  933 | Hüllkurvensteuerung: Mindestgrenze für Hochdruck des Verdichters 3 „Wie oben, für den Verdichter Nr.3“. M CO | Hüllkurvensteuerung: Mindestgrenze für Hochdruck des Verdichters 3 „Wie oben, für den Verdichter Nr.3“. M CO | Envelope control: Mindestgrenze für Hochdruck compressors 3 „Wie oben, für compressor Nr.3“. M CO | Envelope control: Mindestgrenze für Hochdruck compresseurs 3 „Wie oben, für compresseur Nr.3“. M CO | Envelope control: Mindestgrenze für Hochdruck compressores 3 „Wie oben, für compressore Nr.3“. M CO
  934 | Hüllkurvensteuerung: Mindestgrenze für Hochdruck des Verdichters 4 „Wie oben, für den Verdichter Nr.4“. M CO | Hüllkurvensteuerung: Mindestgrenze für Hochdruck des Verdichters 4 „Wie oben, für den Verdichter Nr.4“. M CO | Envelope control: Mindestgrenze für Hochdruck compressors 4 „Wie oben, für compressor Nr.4“. M CO | Envelope control: Mindestgrenze für Hochdruck compresseurs 4 „Wie oben, für compresseur Nr.4“. M CO | Envelope control: Mindestgrenze für Hochdruck compressores 4 „Wie oben, für compressore Nr.4“. M CO
  935 | Hüllkurvensteuerung: Mindestgrenze für Hochdruck des Verdichters 5 „Wie oben, für den Verdichter Nr. 5“. M CO | Hüllkurvensteuerung: Mindestgrenze für Hochdruck des Verdichters 5 „Wie oben, für den Verdichter Nr. 5“. M CO | Envelope control: Mindestgrenze für Hochdruck compressors 5 „Wie oben, für compressor Nr. 5“. M CO | Envelope control: Mindestgrenze für Hochdruck compresseurs 5 „Wie oben, für compresseur Nr. 5“. M CO | Envelope control: Mindestgrenze für Hochdruck compressores 5 „Wie oben, für compressore Nr. 5“. M CO
  936 | Hüllkurvensteuerung: Mindestgrenze für Hochdruck des Verdichters 6 „Wie oben, für den Verdichter Nr. 6“. M CO | Hüllkurvensteuerung: Mindestgrenze für Hochdruck des Verdichters 6 „Wie oben, für den Verdichter Nr. 6“. M CO | Envelope control: Mindestgrenze für Hochdruck compressors 6 „Wie oben, für compressor Nr. 6“. M CO | Envelope control: Mindestgrenze für Hochdruck compresseurs 6 „Wie oben, für compresseur Nr. 6“. M CO | Envelope control: Mindestgrenze für Hochdruck compressores 6 „Wie oben, für compressore Nr. 6“. M CO
  937 | Hüllkurvensteuerung: Mindestgrenze für Hochdruck des Verdichters 7 „Wie oben, für den Verdichter Nr. 7“. M CO | Hüllkurvensteuerung: Mindestgrenze für Hochdruck des Verdichters 7 „Wie oben, für den Verdichter Nr. 7“. M CO | Envelope control: Mindestgrenze für Hochdruck compressors 7 „Wie oben, für compressor Nr. 7“. M CO | Envelope control: Mindestgrenze für Hochdruck compresseurs 7 „Wie oben, für compresseur Nr. 7“. M CO | Envelope control: Mindestgrenze für Hochdruck compressores 7 „Wie oben, für compressore Nr. 7“. M CO
  938 | Hüllkurvensteuerung: Mindestgrenze für Hochdruck des Verdichters 8 „Wie oben, für den Verdichter Nr. 8“. M CO | Hüllkurvensteuerung: Mindestgrenze für Hochdruck des Verdichters 8 „Wie oben, für den Verdichter Nr. 8“. M CO | Envelope control: Mindestgrenze für Hochdruck compressors 8 „Wie oben, für compressor Nr. 8“. M CO | Envelope control: Mindestgrenze für Hochdruck compresseurs 8 „Wie oben, für compresseur Nr. 8“. M CO | Envelope control: Mindestgrenze für Hochdruck compressores 8 „Wie oben, für compressore Nr. 8“. M CO
  941 | Min. Verdichtungsverhältnis beim Anlaufen des Verdichters 1 | Min. Verdichtungsverhältnis beim Anlaufen des Verdichters 1 | Min. Verdichtungsverhältnis beim Anlaufen compressors 1 | Min. Verdichtungsverhältnis beim Anlaufen compresseurs 1 | Min. Verdichtungsverhältnis beim Anlaufen compressores 1
  942 | Min. Verdichtungsverhältnis beim Anlaufen des Verdichters 2 „Wie oben, für den Verdichter Nr.2“. M CO | Min. Verdichtungsverhältnis beim Anlaufen des Verdichters 2 „Wie oben, für den Verdichter Nr.2“. M CO | Min. Verdichtungsverhältnis beim Anlaufen compressors 2 „Wie oben, für compressor Nr.2“. M CO | Min. Verdichtungsverhältnis beim Anlaufen compresseurs 2 „Wie oben, für compresseur Nr.2“. M CO | Min. Verdichtungsverhältnis beim Anlaufen compressores 2 „Wie oben, für compressore Nr.2“. M CO
  943 | Min. Verdichtungsverhältnis beim Anlaufen des Verdichters 3 „Wie oben, für den Verdichter Nr.3“. M CO | Min. Verdichtungsverhältnis beim Anlaufen des Verdichters 3 „Wie oben, für den Verdichter Nr.3“. M CO | Min. Verdichtungsverhältnis beim Anlaufen compressors 3 „Wie oben, für compressor Nr.3“. M CO | Min. Verdichtungsverhältnis beim Anlaufen compresseurs 3 „Wie oben, für compresseur Nr.3“. M CO | Min. Verdichtungsverhältnis beim Anlaufen compressores 3 „Wie oben, für compressore Nr.3“. M CO
  944 | Min. Verdichtungsverhältnis beim Anlaufen des Verdichters 4 „Wie oben, für den Verdichter Nr.4“. M CO | Min. Verdichtungsverhältnis beim Anlaufen des Verdichters 4 „Wie oben, für den Verdichter Nr.4“. M CO | Min. Verdichtungsverhältnis beim Anlaufen compressors 4 „Wie oben, für compressor Nr.4“. M CO | Min. Verdichtungsverhältnis beim Anlaufen compresseurs 4 „Wie oben, für compresseur Nr.4“. M CO | Min. Verdichtungsverhältnis beim Anlaufen compressores 4 „Wie oben, für compressore Nr.4“. M CO
  945 | Min. Verdichtungsverhältnis beim Anlaufen des Verdichters 5 „Wie oben, für den Verdichter Nr. 5“. M CO | Min. Verdichtungsverhältnis beim Anlaufen des Verdichters 5 „Wie oben, für den Verdichter Nr. 5“. M CO | Min. Verdichtungsverhältnis beim Anlaufen compressors 5 „Wie oben, für compressor Nr. 5“. M CO | Min. Verdichtungsverhältnis beim Anlaufen compresseurs 5 „Wie oben, für compresseur Nr. 5“. M CO | Min. Verdichtungsverhältnis beim Anlaufen compressores 5 „Wie oben, für compressore Nr. 5“. M CO
  946 | Min. Verdichtungsverhältnis beim Anlaufen des Verdichters 6 „Wie oben, für den Verdichter Nr. 6“. M CO | Min. Verdichtungsverhältnis beim Anlaufen des Verdichters 6 „Wie oben, für den Verdichter Nr. 6“. M CO | Min. Verdichtungsverhältnis beim Anlaufen compressors 6 „Wie oben, für compressor Nr. 6“. M CO | Min. Verdichtungsverhältnis beim Anlaufen compresseurs 6 „Wie oben, für compresseur Nr. 6“. M CO | Min. Verdichtungsverhältnis beim Anlaufen compressores 6 „Wie oben, für compressore Nr. 6“. M CO
  947 | Min. Verdichtungsverhältnis beim Anlaufen des Verdichters 7 „Wie oben, für den Verdichter Nr. 7“. M CO | Min. Verdichtungsverhältnis beim Anlaufen des Verdichters 7 „Wie oben, für den Verdichter Nr. 7“. M CO | Min. Verdichtungsverhältnis beim Anlaufen compressors 7 „Wie oben, für compressor Nr. 7“. M CO | Min. Verdichtungsverhältnis beim Anlaufen compresseurs 7 „Wie oben, für compresseur Nr. 7“. M CO | Min. Verdichtungsverhältnis beim Anlaufen compressores 7 „Wie oben, für compressore Nr. 7“. M CO
  948 | Min. Verdichtungsverhältnis beim Anlaufen des Verdichters 8 „Wie oben, für den Verdichter Nr. 8“. M CO | Min. Verdichtungsverhältnis beim Anlaufen des Verdichters 8 „Wie oben, für den Verdichter Nr. 8“. M CO | Min. Verdichtungsverhältnis beim Anlaufen compressors 8 „Wie oben, für compressor Nr. 8“. M CO | Min. Verdichtungsverhältnis beim Anlaufen compresseurs 8 „Wie oben, für compresseur Nr. 8“. M CO | Min. Verdichtungsverhältnis beim Anlaufen compressores 8 „Wie oben, für compressore Nr. 8“. M CO
  951 | Trennung HGBP -Ventil des Verdichters 1 | Trennung HGBP -Ventil des Verdichters 1 | Disconnection HGBP -Ventil compressors 1 | Disconnection HGBP -Ventil compresseurs 1 | Disconnection HGBP -Ventil compressores 1
  952 | Trennung HGBP -Ventil des Verdichters 2 „Wie oben, für den Verdichter Nr.2“. S CO | Trennung HGBP -Ventil des Verdichters 2 „Wie oben, für den Verdichter Nr.2“. S CO | Disconnection HGBP -Ventil compressors 2 „Wie oben, für compressor Nr.2“. S CO | Disconnection HGBP -Ventil compresseurs 2 „Wie oben, für compresseur Nr.2“. S CO | Disconnection HGBP -Ventil compressores 2 „Wie oben, für compressore Nr.2“. S CO
  953 | Trennung HGBP -Ventil des Verdichters 3 „Wie oben, für den Verdichter Nr.3“. S CO | Trennung HGBP -Ventil des Verdichters 3 „Wie oben, für den Verdichter Nr.3“. S CO | Disconnection HGBP -Ventil compressors 3 „Wie oben, für compressor Nr.3“. S CO | Disconnection HGBP -Ventil compresseurs 3 „Wie oben, für compresseur Nr.3“. S CO | Disconnection HGBP -Ventil compressores 3 „Wie oben, für compressore Nr.3“. S CO
  954 | Trennung HGBP -Ventil des Verdichters 4 „Wie oben, für den Verdichter Nr.4“. S CO | Trennung HGBP -Ventil des Verdichters 4 „Wie oben, für den Verdichter Nr.4“. S CO | Disconnection HGBP -Ventil compressors 4 „Wie oben, für compressor Nr.4“. S CO | Disconnection HGBP -Ventil compresseurs 4 „Wie oben, für compresseur Nr.4“. S CO | Disconnection HGBP -Ventil compressores 4 „Wie oben, für compressore Nr.4“. S CO
  960 | Trennung thermal meter | Trennung thermal meter | Disconnection thermal meter | Disconnection thermal meter | Disconnection thermal meter
  961 | Offline Driver erste Stufe Nr.5 | Offline Driver erste Stufe Nr.5 | Offline Driver erste Stufe Nr.5 | Offline Driver erste Stufe Nr.5 | Offline Driver erste Stufe Nr.5
  962 | Offline Driver erste Stufe Nr.6 „Wie oben, für den Verdichter 6“. A CI | Offline Driver erste Stufe Nr.6 „Wie oben, für den Verdichter 6“. A CI | Offline Driver erste Stufe Nr.6 „Wie oben, für compressor 6“. A CI | Offline Driver erste Stufe Nr.6 „Wie oben, für compresseur 6“. A CI | Offline Driver erste Stufe Nr.6 „Wie oben, für compressore 6“. A CI
  963 | Offline Driver erste Stufe Nr.7 „Wie oben, für den Verdichter 7“. A CI | Offline Driver erste Stufe Nr.7 „Wie oben, für den Verdichter 7“. A CI | Offline Driver erste Stufe Nr.7 „Wie oben, für compressor 7“. A CI | Offline Driver erste Stufe Nr.7 „Wie oben, für compresseur 7“. A CI | Offline Driver erste Stufe Nr.7 „Wie oben, für compressore 7“. A CI
  964 | Offline Driver erste Stufe Nr.8 „Wie oben, für den Verdichter 8“. A CI | Offline Driver erste Stufe Nr.8 „Wie oben, für den Verdichter 8“. A CI | Offline Driver erste Stufe Nr.8 „Wie oben, für compressor 8“. A CI | Offline Driver erste Stufe Nr.8 „Wie oben, für compresseur 8“. A CI | Offline Driver erste Stufe Nr.8 „Wie oben, für compressore 8“. A CI
  965 | Trennung ATS | Trennung ATS | Disconnection ATS | Disconnection ATS | Disconnection ATS
  966 | Trennung Touch HT -Zone Meldet die Trennung des Touch -Thermostaten der Zone HT. S GR | Trennung Touch HT -Zone Meldet die Trennung des Touch -Thermostaten der Zone HT. S GR | Disconnection Touch HT -Zone Meldet Trennung Touch -Thermostaten Zone HT. S GR | Disconnection Touch HT -Zone Meldet Trennung Touch -Thermostaten Zone HT. S GR | Disconnection Touch HT -Zone Meldet Trennung Touch -Thermostaten Zone HT. S GR
  967 | Trennung Touch LT -Zone Meldet die Trennung des Touch -Thermostaten der Zone LT. S GR | Trennung Touch LT -Zone Meldet die Trennung des Touch -Thermostaten der Zone LT. S GR | Disconnection Touch LT -Zone Meldet Trennung Touch -Thermostaten Zone LT. S GR | Disconnection Touch LT -Zone Meldet Trennung Touch -Thermostaten Zone LT. S GR | Disconnection Touch LT -Zone Meldet Trennung Touch -Thermostaten Zone LT. S GR
  968 | Verhinderung von Stillstand des Verdichters Meldet die Zwangsabschaltung des Inverter - Verdichters und seines Kreislaufs, um einen Stillstand aufgrund eines zu hohen Stromverbrauchs zu verhindern. M CI | Verhinderung von Stillstand des Verdichters Meldet die Zwangsabschaltung des Inverter - Verdichters und seines Kreislaufs, um einen Stillstand aufgrund eines zu hohen Stromverbrauchs zu verhindern. M CI | Verhinderung von Stillstand compressors Meldet Zwangsabschaltung inverter - compressors und seines circuits, um einen Stillstand aufgrund eines zu hohen Stromverbrauchs zu verhindern. M CI | Verhinderung von Stillstand compresseurs Meldet Zwangsabschaltung variateur - compresseurs und seines circuits, um einen Stillstand aufgrund eines zu hohen Stromverbrauchs zu verhindern. M CI | Verhinderung von Stillstand compressores Meldet Zwangsabschaltung inverter - compressores und seines circuitos, um einen Stillstand aufgrund eines zu hohen Stromverbrauchs zu verhindern. M CI
  969 | Hohe Außenlufttemperatur Meldet, dass das Gerät bei einer zu hohen Außentemperatur betrieben wird. Die Kontrolle erfolgt auch bei ausgeschalteten Verdichtern. S-M U STG0200 | Hohe Außenlufttemperatur Meldet, dass das Gerät bei einer zu hohen Außentemperatur betrieben wird. Die Kontrolle erfolgt auch bei ausgeschalteten Verdichtern. S-M U STG0200 | Hohe outdoor air temperature Meldet, dass Gerät bei einer zu hohen Außentemperatur betrieben wird. Kontrolle erfolgt auch bei ausgeschalteten compressorn. S-M U STG0200 | Hohe température extérieure Meldet, dass Gerät bei einer zu hohen Außentemperatur betrieben wird. Kontrolle erfolgt auch bei ausgeschalteten compresseurn. S-M U STG0200 | Hohe temperatura aria esterna Meldet, dass Gerät bei einer zu hohen Außentemperatur betrieben wird. Kontrolle erfolgt auch bei ausgeschalteten compressoren. S-M U STG0200
  970 | Geringer Wassergehalt bei der Wärmerückgewinnung. Meldet einen Wassermangel im Wasserkreislauf für die Wärmerückgewinnung. Dieser Mangel führt zu plötzlichen Wechseln der Betriebsart der Kreisläufe, wodurch die Ventile des Kältemittelkreislaufs beschädigt werden können. S-M U | Geringer Wassergehalt bei der Wärmerückgewinnung. Meldet einen Wassermangel im Wasserkreislauf für die Wärmerückgewinnung. Dieser Mangel führt zu plötzlichen Wechseln der Betriebsart der Kreisläufe, wodurch die Ventile des Kältemittelkreislaufs beschädigt werden können. S-M U | Geringer Wassergehalt bei heat recovery. Meldet einen Wassermangel im Wassercircuit für heat recovery. Dieser Mangel führt zu plötzlichen Wechseln Betriebsart Kreisläufe, wodurch Ventile Kältemittelcircuits beschädigt werden können. S-M U | Geringer Wassergehalt bei récupération de chaleur. Meldet einen Wassermangel im Wassercircuit für récupération de chaleur. Dieser Mangel führt zu plötzlichen Wechseln Betriebsart Kreisläufe, wodurch Ventile Kältemittelcircuits beschädigt werden können. S-M U | Geringer Wassergehalt bei recupero di calore. Meldet einen Wassermangel im Wassercircuito für recupero di calore. Dieser Mangel führt zu plötzlichen Wechseln Betriebsart Kreisläufe, wodurch Ventile Kältemittelcircuitos beschädigt werden können. S-M U
  971 | Wartung von Gassensor | Wartung von Gassensor | Maintenance von Gassensor | Maintenance von Gassensor | Maintenance von Gassensor
  972 | Anomalie Low Lift-Pumpe 1 | Anomalie Low Lift-Pumpe 1 | Anomalie Low Lift-pump 1 | Anomalie Low Lift-pompe 1 | Anomalie Low Lift-pompa 1
  973 | Anomalie Low Lift-Pumpe 2 | Anomalie Low Lift-Pumpe 2 | Anomalie Low Lift-pump 2 | Anomalie Low Lift-pompe 2 | Anomalie Low Lift-pompa 2
  974 | Alarm niedrige Temperatur Trockenkühler Das Signal erscheint bei Geräten, die mit einem Dry Cooler ausgestattet sind, wenn die Temperatur der Installationsumgebung des Dry Cooler niedriger als der eingestellte Sollwert ist. A U | Alarm niedrige Temperatur Trockenkühler Das Signal erscheint bei Geräten, die mit einem Dry Cooler ausgestattet sind, wenn die Temperatur der Installationsumgebung des Dry Cooler niedriger als der eingestellte Sollwert ist. A U | Alarm Low temperature Trockenkühler Signal erscheint bei Geräten, mit einem Dry Cooler ausgestattet sind, wenn Temperatur Installationsumgebung Dry Cooler niedriger als eingestellte Sollwert ist. A U | Alarm Low temperature Trockenkühler Signal erscheint bei Geräten, mit einem Dry Cooler ausgestattet sind, wenn Temperatur Installationsumgebung Dry Cooler niedriger als eingestellte Sollwert ist. A U | Alarm Low temperature Trockenkühler Signal erscheint bei Geräten, mit einem Dry Cooler ausgestattet sind, wenn Temperatur Installationsumgebung Dry Cooler niedriger als eingestellte Sollwert ist. A U
  975 | Störung Trockenkühler Das Signal erscheint bei Geräten, die mit einem Dry Cooler ausgestattet sind, wenn der thermische Schutz der Ventilatoren oder die entsprechende Pumpe (falls vorhanden) eingreift. M U | Störung Trockenkühler Das Signal erscheint bei Geräten, die mit einem Dry Cooler ausgestattet sind, wenn der thermische Schutz der Ventilatoren oder die entsprechende Pumpe (falls vorhanden) eingreift. M U | Fault Trockenkühler Signal erscheint bei Geräten, mit einem Dry Cooler ausgestattet sind, wenn thermische Schutz fanen oder entsprechende pump (falls vorhanden) eingreift. M U | Fault Trockenkühler Signal erscheint bei Geräten, mit einem Dry Cooler ausgestattet sind, wenn thermische Schutz ventilateuren oder entsprechende pompe (falls vorhanden) eingreift. M U | Fault Trockenkühler Signal erscheint bei Geräten, mit einem Dry Cooler ausgestattet sind, wenn thermische Schutz ventilatoreen oder entsprechende pompa (falls vorhanden) eingreift. M U
  5001 | Störung Betriebsmodus -Änderung Alarm, der eine Störung während der erzwungenen Änderung des Betriebsmodus der Einheit meldet, wenn sich der Betriebsmodus der Anlage ändert. Der Alarm wird aktiviert, wenn die Forcierung innerhalb der durch den Parameter festgelegten maximalen Zeit nicht erfolgreich umgesetzt wird. M GR GRP0126 | Störung Betriebsmodus -Änderung Alarm, der eine Störung während der erzwungenen Änderung des Betriebsmodus der Einheit meldet, wenn sich der Betriebsmodus der Anlage ändert. Der Alarm wird aktiviert, wenn die Forcierung innerhalb der durch den Parameter festgelegten maximalen Zeit nicht erfolgreich umgesetzt wird. M GR GRP0126 | Fault Betriebsmodus -Änderung Alarm, eine Störung während erzwungenen Änderung Betriebsmodus unit meldet, wenn sich Betriebsmodus system ändert. Alarm wird aktiviert, wenn Forcierung innerhalb durch Parameter festgelegten maximalen Zeit nicht erfolgreich umgesetzt wird. M GR GRP0126 | Fault Betriebsmodus -Änderung Alarm, eine Störung während erzwungenen Änderung Betriebsmodus unité meldet, wenn sich Betriebsmodus installation ändert. Alarm wird aktiviert, wenn Forcierung innerhalb durch Parameter festgelegten maximalen Zeit nicht erfolgreich umgesetzt wird. M GR GRP0126 | Fault Betriebsmodus -Änderung Alarm, eine Störung während erzwungenen Änderung Betriebsmodus unità meldet, wenn sich Betriebsmodus impianto ändert. Alarm wird aktiviert, wenn Forcierung innerhalb durch Parameter festgelegten maximalen Zeit nicht erfolgreich umgesetzt wird. M GR GRP0126
  5005 | Fehler Durchschnitt Wassertemp.fühler Eingang Fehler im Durchschnitt der von den Sonden aller in der Gruppe vorhandenen Einheiten gemessenen Eingangstemperaturwerte. A GR | Fehler Durchschnitt Wassertemp.fühler Eingang Fehler im Durchschnitt der von den Sonden aller in der Gruppe vorhandenen Einheiten gemessenen Eingangstemperaturwerte. A GR | Fehler Durchschnitt Wassertemp.sensor inlet Fehler im Durchschnitt von Sonden aller in Gruppe vorhandenen uniten gemessenen inletstemperaturwerte. A GR | Fehler Durchschnitt Wassertemp.sonde entrée Fehler im Durchschnitt von Sonden aller in Gruppe vorhandenen unitéen gemessenen entréestemperaturwerte. A GR | Fehler Durchschnitt Wassertemp.sensore ingresso Fehler im Durchschnitt von Sonden aller in Gruppe vorhandenen unitàen gemessenen ingressostemperaturwerte. A GR
  5006 | Fehler Durchschnitt Wassertemp.fühler Ausgang Fehler im Durchschnitt der von den Sonden aller in der Gruppe vorhandenen Einheiten gemessenen Austrittstemperaturwerte. A GR | Fehler Durchschnitt Wassertemp.fühler Ausgang Fehler im Durchschnitt der von den Sonden aller in der Gruppe vorhandenen Einheiten gemessenen Austrittstemperaturwerte. A GR | Fehler Durchschnitt Wassertemp.sensor outlet Fehler im Durchschnitt von Sonden aller in Gruppe vorhandenen uniten gemessenen Austrittstemperaturwerte. A GR | Fehler Durchschnitt Wassertemp.sonde sortie Fehler im Durchschnitt von Sonden aller in Gruppe vorhandenen unitéen gemessenen Austrittstemperaturwerte. A GR | Fehler Durchschnitt Wassertemp.sensore uscita Fehler im Durchschnitt von Sonden aller in Gruppe vorhandenen unitàen gemessenen Austrittstemperaturwerte. A GR
  5050 | Fehler Durchschnitt Außentemperaturfühler Fehler im Durchschnitt der von den Sonden aller in der Gruppe vorhandenen Einheiten gemessenen Außentemperaturwerte. A GR | Fehler Durchschnitt Außentemperaturfühler Fehler im Durchschnitt der von den Sonden aller in der Gruppe vorhandenen Einheiten gemessenen Außentemperaturwerte. A GR | Fehler Durchschnitt Außentemperature sensor Fehler im Durchschnitt von Sonden aller in Gruppe vorhandenen uniten gemessenen Außentemperaturwerte. A GR | Fehler Durchschnitt Außensonde de température Fehler im Durchschnitt von Sonden aller in Gruppe vorhandenen unitéen gemessenen Außentemperaturwerte. A GR | Fehler Durchschnitt Außensensore di temperatura Fehler im Durchschnitt von Sonden aller in Gruppe vorhandenen unitàen gemessenen Außentemperaturwerte. A GR
  5080 | Schutzschalter Anlagenpumpe Meldet die Überhitzung der Anlagenpumpe. M GR | Schutzschalter Anlagenpumpe Meldet die Überhitzung der Anlagenpumpe. M GR | Protection switch plant pump Meldet Überhitzung plant pump. M GR | Protection switch pompe d’installation Meldet Überhitzung pompe d’installation. M GR | Protection switch pompa impianto Meldet Überhitzung pompa impianto. M GR
  5100 | Gruppen- Steuermodul VPF nicht angeschlossen Das Modul, das den Wasserdurchfluss der Anlage steuert, ist nicht angeschlossen. Die Störung an der Benutzerschnittstelle des Moduls überprüfen. A GR | Gruppen- Steuermodul VPF nicht angeschlossen Das Modul, das den Wasserdurchfluss der Anlage steuert, ist nicht angeschlossen. Die Störung an der Benutzerschnittstelle des Moduls überprüfen. A GR | Gruppen- Steuermodul VPF nicht angeschlossen Modul, Wasserdurchfluss system steuert, ist nicht angeschlossen. Störung an Benutzerschnittstelle Moduls überprüfen. A GR | Gruppen- Steuermodul VPF nicht angeschlossen Modul, Wasserdurchfluss installation steuert, ist nicht angeschlossen. Störung an Benutzerschnittstelle Moduls überprüfen. A GR | Gruppen- Steuermodul VPF nicht angeschlossen Modul, Wasserdurchfluss impianto steuert, ist nicht angeschlossen. Störung an Benutzerschnittstelle Moduls überprüfen. A GR
  5101 | Störung Gruppen -Steuermodul VPF Störung am Modul, das den Wasserdurchfluss der Anlage steuert. Die Störung an der Benutzerschnittstelle des Moduls überprüfen. A GR | Störung Gruppen -Steuermodul VPF Störung am Modul, das den Wasserdurchfluss der Anlage steuert. Die Störung an der Benutzerschnittstelle des Moduls überprüfen. A GR | Fault Gruppen -Steuermodul VPF Störung am Modul, Wasserdurchfluss system steuert. Störung an Benutzerschnittstelle Moduls überprüfen. A GR | Fault Gruppen -Steuermodul VPF Störung am Modul, Wasserdurchfluss installation steuert. Störung an Benutzerschnittstelle Moduls überprüfen. A GR | Fault Gruppen -Steuermodul VPF Störung am Modul, Wasserdurchfluss impianto steuert. Störung an Benutzerschnittstelle Moduls überprüfen. A GR
  5120 | Unterbrechung dynamischer Setpoint Unterbrechung der dynamischen Verwaltung des Gruppen- Setpoints. Überprüfen, ob evtl. im KIPLan -Netzwerk Unterbrechungen in der Verbindung auftreten. A GR | Unterbrechung dynamischer Setpoint Unterbrechung der dynamischen Verwaltung des Gruppen- Setpoints. Überprüfen, ob evtl. im KIPLan -Netzwerk Unterbrechungen in der Verbindung auftreten. A GR | Unterbrechung dynamischer Setpoint Unterbrechung dynamischen Verwaltung Gruppen- Setpoints. Überprüfen, ob evtl. im KIPLan -Netzwerk Unterbrechungen in Verbindung auftreten. A GR | Unterbrechung dynamischer Setpoint Unterbrechung dynamischen Verwaltung Gruppen- Setpoints. Überprüfen, ob evtl. im KIPLan -Netzwerk Unterbrechungen in Verbindung auftreten. A GR | Unterbrechung dynamischer Setpoint Unterbrechung dynamischen Verwaltung Gruppen- Setpoints. Überprüfen, ob evtl. im KIPLan -Netzwerk Unterbrechungen in Verbindung auftreten. A GR
  5201 | Fehler Fühler 1 Gruppe Fehler Fühler 1 der Gruppen -Reglereinheit. Die vom Fühler 1 gemessenen Werte liegen außerhalb der Grenzwerte. A GR | Fehler Fühler 1 Gruppe Fehler Fühler 1 der Gruppen -Reglereinheit. Die vom Fühler 1 gemessenen Werte liegen außerhalb der Grenzwerte. A GR | Fehler sensor 1 Gruppe Fehler sensor 1 Gruppen -Reglerunit. vom sensor 1 gemessenen Werte liegen außerhalb Grenzwerte. A GR | Fehler sonde 1 Gruppe Fehler sonde 1 Gruppen -Reglerunité. vom sonde 1 gemessenen Werte liegen außerhalb Grenzwerte. A GR | Fehler sensore 1 Gruppe Fehler sensore 1 Gruppen -Reglerunità. vom sensore 1 gemessenen Werte liegen außerhalb Grenzwerte. A GR
  5202 | Fehler Fühler 2 Gruppe „analog, wie oben“. A GR | Fehler Fühler 2 Gruppe „analog, wie oben“. A GR | Fehler sensor 2 Gruppe „analog, wie oben“. A GR | Fehler sonde 2 Gruppe „analog, wie oben“. A GR | Fehler sensore 2 Gruppe „analog, wie oben“. A GR
  5203 | Fehler Fühler 3 Gruppe „analog, wie oben“. A GR | Fehler Fühler 3 Gruppe „analog, wie oben“. A GR | Fehler sensor 3 Gruppe „analog, wie oben“. A GR | Fehler sonde 3 Gruppe „analog, wie oben“. A GR | Fehler sensore 3 Gruppe „analog, wie oben“. A GR
  5204 | Fehler Fühler 4 Gruppe „analog, wie oben“. A GR | Fehler Fühler 4 Gruppe „analog, wie oben“. A GR | Fehler sensor 4 Gruppe „analog, wie oben“. A GR | Fehler sonde 4 Gruppe „analog, wie oben“. A GR | Fehler sensore 4 Gruppe „analog, wie oben“. A GR
  5205 | Fehler Fühler 5 Gruppe „analog, wie oben“. A GR | Fehler Fühler 5 Gruppe „analog, wie oben“. A GR | Fehler sensor 5 Gruppe „analog, wie oben“. A GR | Fehler sonde 5 Gruppe „analog, wie oben“. A GR | Fehler sensore 5 Gruppe „analog, wie oben“. A GR
  5206 | Fehler Fühler 6 Gruppe „analog, wie oben“. A GR | Fehler Fühler 6 Gruppe „analog, wie oben“. A GR | Fehler sensor 6 Gruppe „analog, wie oben“. A GR | Fehler sonde 6 Gruppe „analog, wie oben“. A GR | Fehler sensore 6 Gruppe „analog, wie oben“. A GR
  5207 | Fehler Fühler 7 Gruppe „analog, wie oben“. A GR | Fehler Fühler 7 Gruppe „analog, wie oben“. A GR | Fehler sensor 7 Gruppe „analog, wie oben“. A GR | Fehler sonde 7 Gruppe „analog, wie oben“. A GR | Fehler sensore 7 Gruppe „analog, wie oben“. A GR
  5208 | Fehler Fühler 8 Gruppe „analog, wie oben“. A GR | Fehler Fühler 8 Gruppe „analog, wie oben“. A GR | Fehler sensor 8 Gruppe „analog, wie oben“. A GR | Fehler sonde 8 Gruppe „analog, wie oben“. A GR | Fehler sensore 8 Gruppe „analog, wie oben“. A GR
  5209 | Fehler Fühler 9 Gruppe „analog, wie oben“. A GR | Fehler Fühler 9 Gruppe „analog, wie oben“. A GR | Fehler sensor 9 Gruppe „analog, wie oben“. A GR | Fehler sonde 9 Gruppe „analog, wie oben“. A GR | Fehler sensore 9 Gruppe „analog, wie oben“. A GR
  5210 | Fehler Fühler 10 Gruppe „analog, wie oben“. A GR | Fehler Fühler 10 Gruppe „analog, wie oben“. A GR | Fehler sensor 10 Gruppe „analog, wie oben“. A GR | Fehler sonde 10 Gruppe „analog, wie oben“. A GR | Fehler sensore 10 Gruppe „analog, wie oben“. A GR
  5301 | Offline Einheit 1 | Offline Einheit 1 | Offline unit 1 | Offline unité 1 | Offline unità 1
  5302 | Offline Einheit 2 „analog, wie oben für Einheit 2“. A GR | Offline Einheit 2 „analog, wie oben für Einheit 2“. A GR | Offline unit 2 „analog, wie oben für unit 2“. A GR | Offline unité 2 „analog, wie oben für unité 2“. A GR | Offline unità 2 „analog, wie oben für unità 2“. A GR
  5303 | Offline Einheit 3 „analog, wie oben für Einheit 3“. A GR | Offline Einheit 3 „analog, wie oben für Einheit 3“. A GR | Offline unit 3 „analog, wie oben für unit 3“. A GR | Offline unité 3 „analog, wie oben für unité 3“. A GR | Offline unità 3 „analog, wie oben für unità 3“. A GR
  5304 | Offline Einheit 4 „analog, wie oben für Einheit 4“. A GR | Offline Einheit 4 „analog, wie oben für Einheit 4“. A GR | Offline unit 4 „analog, wie oben für unit 4“. A GR | Offline unité 4 „analog, wie oben für unité 4“. A GR | Offline unità 4 „analog, wie oben für unità 4“. A GR
  5305 | Offline Einheit 5 „analog, wie oben für Einheit 5“. A GR | Offline Einheit 5 „analog, wie oben für Einheit 5“. A GR | Offline unit 5 „analog, wie oben für unit 5“. A GR | Offline unité 5 „analog, wie oben für unité 5“. A GR | Offline unità 5 „analog, wie oben für unità 5“. A GR
  5306 | Offline Einheit 6 „analog, wie oben für Einheit 6“. A GR | Offline Einheit 6 „analog, wie oben für Einheit 6“. A GR | Offline unit 6 „analog, wie oben für unit 6“. A GR | Offline unité 6 „analog, wie oben für unité 6“. A GR | Offline unità 6 „analog, wie oben für unità 6“. A GR
  5307 | Offline Einheit 7 „analog, wie oben für Einheit 7“. A GR | Offline Einheit 7 „analog, wie oben für Einheit 7“. A GR | Offline unit 7 „analog, wie oben für unit 7“. A GR | Offline unité 7 „analog, wie oben für unité 7“. A GR | Offline unità 7 „analog, wie oben für unità 7“. A GR
  5308 | Offline Einheit 8 „analog, wie oben für Einheit 8“. A GR | Offline Einheit 8 „analog, wie oben für Einheit 8“. A GR | Offline unit 8 „analog, wie oben für unit 8“. A GR | Offline unité 8 „analog, wie oben für unité 8“. A GR | Offline unità 8 „analog, wie oben für unità 8“. A GR
  5350 | Offline KIPlink Master KIPlink für den Datenaustausch zwischen Außen - und Innengeräten ist nicht angeschlossen. Die seriellen Anschlüsse überprüfen. A GR | Offline KIPlink Master KIPlink für den Datenaustausch zwischen Außen - und Innengeräten ist nicht angeschlossen. Die seriellen Anschlüsse überprüfen. A GR | Offline KIPlink Master KIPlink für Datenaustausch zwischen Außen - und Innengeräten ist nicht angeschlossen. seriellen Anschlüsse überprüfen. A GR | Offline KIPlink Master KIPlink für Datenaustausch zwischen Außen - und Innengeräten ist nicht angeschlossen. seriellen Anschlüsse überprüfen. A GR | Offline KIPlink Master KIPlink für Datenaustausch zwischen Außen - und Innengeräten ist nicht angeschlossen. seriellen Anschlüsse überprüfen. A GR
  5401 | Störung Einheit 1 Es liegen Alarme aufgrund der Sonden der Gruppe vor, die auf die Einheit 1 zurückgeführt werden können. A GR | Störung Einheit 1 Es liegen Alarme aufgrund der Sonden der Gruppe vor, die auf die Einheit 1 zurückgeführt werden können. A GR | Fault unit 1 Es liegen Alarme aufgrund Sonden Gruppe vor, auf unit 1 zurückgeführt werden können. A GR | Fault unité 1 Es liegen Alarme aufgrund Sonden Gruppe vor, auf unité 1 zurückgeführt werden können. A GR | Fault unità 1 Es liegen Alarme aufgrund Sonden Gruppe vor, auf unità 1 zurückgeführt werden können. A GR
  5402 | Störung Einheit 2 „analog, wie oben für Einheit 2“. A GR | Störung Einheit 2 „analog, wie oben für Einheit 2“. A GR | Fault unit 2 „analog, wie oben für unit 2“. A GR | Fault unité 2 „analog, wie oben für unité 2“. A GR | Fault unità 2 „analog, wie oben für unità 2“. A GR
  5403 | Störung Einheit 3 „analog, wie oben für Einheit 3“. A GR | Störung Einheit 3 „analog, wie oben für Einheit 3“. A GR | Fault unit 3 „analog, wie oben für unit 3“. A GR | Fault unité 3 „analog, wie oben für unité 3“. A GR | Fault unità 3 „analog, wie oben für unità 3“. A GR
  5404 | Störung Einheit 4 „analog, wie oben für Einheit 4“. A GR | Störung Einheit 4 „analog, wie oben für Einheit 4“. A GR | Fault unit 4 „analog, wie oben für unit 4“. A GR | Fault unité 4 „analog, wie oben für unité 4“. A GR | Fault unità 4 „analog, wie oben für unità 4“. A GR
  5405 | Störung Einheit 5 „analog, wie oben für Einheit 5“. A GR | Störung Einheit 5 „analog, wie oben für Einheit 5“. A GR | Fault unit 5 „analog, wie oben für unit 5“. A GR | Fault unité 5 „analog, wie oben für unité 5“. A GR | Fault unità 5 „analog, wie oben für unità 5“. A GR
  5406 | Störung Einheit 6 „analog, wie oben für Einheit 6“. A GR | Störung Einheit 6 „analog, wie oben für Einheit 6“. A GR | Fault unit 6 „analog, wie oben für unit 6“. A GR | Fault unité 6 „analog, wie oben für unité 6“. A GR | Fault unità 6 „analog, wie oben für unità 6“. A GR
  5407 | Störung Einheit 7 „analog, wie oben für Einheit 7“. A GR | Störung Einheit 7 „analog, wie oben für Einheit 7“. A GR | Fault unit 7 „analog, wie oben für unit 7“. A GR | Fault unité 7 „analog, wie oben für unité 7“. A GR | Fault unità 7 „analog, wie oben für unità 7“. A GR
  5408 | Störung Einheit 8 „analog, wie oben für Einheit 8“. A GR ( ** ):Für die spezifischen Alarmereignisse einiger Inverter für Verdichter ist eine Codierung vorgesehen, die das vom Inverter erzeugte Ereignis angibt, welches den Alarm in der Steuerung W3000+ ausgelöst hat. Für die vollständige Liste der spezifischen Alarmcodes wird auf die folgenden Alarmtabellen der Inverter verwiesen. | Störung Einheit 8 „analog, wie oben für Einheit 8“. A GR ( ** ):Für die spezifischen Alarmereignisse einiger Inverter für Verdichter ist eine Codierung vorgesehen, die das vom Inverter erzeugte Ereignis angibt, welches den Alarm in der Steuerung W3000+ ausgelöst hat. Für die vollständige Liste der spezifischen Alarmcodes wird auf die folgenden Alarmtabellen der Inverter verwiesen. | Fault unit 8 „analog, wie oben für unit 8“. A GR ( ** ):Für spezifischen Alarmereignisse einiger inverter für compressor ist eine Codierung vorgesehen, vom inverter erzeugte Ereignis angibt, welches Alarm in Steuerung W3000+ ausgelöst hat. Für vollständige Liste spezifischen Alarmcodes wird auf folgenden Alarmtabellen inverter verwiesen. | Fault unité 8 „analog, wie oben für unité 8“. A GR ( ** ):Für spezifischen Alarmereignisse einiger variateur für compresseur ist eine Codierung vorgesehen, vom variateur erzeugte Ereignis angibt, welches Alarm in Steuerung W3000+ ausgelöst hat. Für vollständige Liste spezifischen Alarmcodes wird auf folgenden Alarmtabellen variateur verwiesen. | Fault unità 8 „analog, wie oben für unità 8“. A GR ( ** ):Für spezifischen Alarmereignisse einiger inverter für compressore ist eine Codierung vorgesehen, vom inverter erzeugte Ereignis angibt, welches Alarm in Steuerung W3000+ ausgelöst hat. Für vollständige Liste spezifischen Alarmcodes wird auf folgenden Alarmtabellen inverter verwiesen.
  0 | ??? | ??? | ??? | ??? | ???
  5409 | Freecooling Soll nicht erreicht |  |  |  | 
   |  |  |  |  |  *)

(* text list txtWpReport (id | default | de | en | fr | it)
  60 | Modbus Ausfall |  |  |  | 
   |  |  |  |  |  *)
